(* IEC 61131-3 sources: verifaps-lib/flycheck/src/test/resources, 2 files *)

(* ---- testoo.st ---- *)
class A implements Z

method override MM
  var_input i : bool; end_var
end_method

end_class

interface Z

method MM
end_method

method error_body : bool
  error_body:= FALSE;
end_method

end_interface

(* ---- test.st ---- *)
FUNCTION b : ABC
VAR
    a : INT;
END_VAR

a := c;
b := a;

END_FUNCTION

FUNCTION e : SINT
VAR
    a : INT;
END_VAR
e := a;
END_FUNCTION
